// TIA Portal V19 export
TYPE "LEXCHANGETRAY_typeHandlingXyzEm_toConstraintRollerReq"
// stored: Access Published
   STRUCT
      transferEnable : Bool;   // 请求抓取
   END_STRUCT;
END_TYPE
